TYPE "GCS7_M_FB55_Data"	// UDT 20550
VERSION : 0.0
  STRUCT
   StCode : INT ;	// State as code 32=StFault 1=StStopped 2=StStarting 3=StStartedWait 4=StStartedF
   InEnableMill1 : BOOL ;	// Enable to run mill 1
   InEnableMill2 : BOOL ;	// Enable to run mill 2
   InDischargeOkMill1 : BOOL ;	// Discharge of mill 1 is ok, starting condition
   InDischargeOkMill2 : BOOL ;	// Discharge of mill 2 is ok, starting condition
   InUsedMill1 : BOOL ;	// Mill 1 is used
   InUsedMill2 : BOOL ;	// Mill 2 is used
   InEnableFeedMill1 : BOOL ;	// Enable feeding mill 1
   InEnableFeedMill2 : BOOL ;	// Enable feeding mill 2
   CmdTick100ms : BOOL ;	// Tick 100 ms to count time (e.g. brake time)
   spare0301 : BOOL ;	//
   CmdNext : BOOL ;	// Pulse to start the next motor in automatic mode
   CmdFaultReset : BOOL ;	// Command to reset fault
   InLocal : BOOL ;	// Local mode, accept all faults
   spare0305 : BOOL ;	//
   spare0306 : BOOL ;	//
   InSeqStop : BOOL ;	// Mill will stop automatically after idling time
   OutFeedingMill1 : BOOL ;	// Mill 1 is feeding
   OutFeedingMill2 : BOOL ;	// Mill 2 is feeding
   OutLoadedMill1 : BOOL ;	// Mill 1 is loaded with product
   OutLoadedMill2 : BOOL ;	// Mill 2 is loaded with product
   OutEmptyingMill1 : BOOL ;	// Mill 1 emptying time t1 is running
   OutEmptyingMill2 : BOOL ;	// Mill 2 emptying time t2 is running
   OutEmptyingDoneMill1 : BOOL ;	// Emptying time done mill 1
   OutEmptyingDoneMill2 : BOOL ;	// Emptying time done mill 2
   StStopped : BOOL ;	// All motors are stopped
   StStarting : BOOL ;	// Not all relevant motors are started
   StStarted : BOOL ;	// All used motors are started
   StStopping : BOOL ;	// Any motor is stopping
   StFault : BOOL ;	// Any relevant element has a fault
   spare0505 : BOOL ;	//
   spare0506 : BOOL ;	//
   spare0507 : BOOL ;	//
   InBrakeMill1 : BOOL ;	// Brake mill 1
   InBrakeMill2 : BOOL ;	// Brake mill 2
   InOutRevMill : BOOL ;	// Mill motors will be started reverse
   InFastMill : BOOL ;	// Mill motors will be started fast
   spare0604 : BOOL ;	//
   spare0605 : BOOL ;	//
   spare0606 : BOOL ;	//
   spare0607 : BOOL ;	//
   InAlarmTempMill1 : BOOL ;	// Temperature alarm mill 1, changing to fault
   InAlarmTempMill2 : BOOL ;	// Temperature alarm mill 2, changing to fault
   spare0702 : BOOL ;	//
   spare0703 : BOOL ;	//
   InpS311Z2 : BOOL ;	// Digital input S311Z2: automatic mode mill 1
   InpS361Z2 : BOOL ;	// Digital input S361Z2: automatic mode mill 2
   InpS311Z2_1 : BOOL ;	// Digital input S311Z2/1: service mode mill 1
   InpS361Z2_1 : BOOL ;	// Digital input S361Z2/1: service mode mill 2
   InpS311Z3 : BOOL ;	// Digital input S311Z3: open cone mill 1
   InpS361Z3 : BOOL ;	// Digital input S361Z3: open cone mill 2
   InpS311Z4 : BOOL ;	// Digital input S311Z4: close cone mill 1
   InpS361Z4 : BOOL ;	// Digital input S361Z4: close cone mill 2
   InpS311Z5 : BOOL ;	// Digital input S311Z5: open haevy-particle gate mill 1
   InpS361Z5 : BOOL ;	// Digital input S361Z5: open haevy-particle gate mill 2
   InpS311Z6 : BOOL ;	// Digital input S311Z6: screen change acknowledge mill 1
   InpS361Z6 : BOOL ;	// Digital input S361Z6: screen change acknowledge mill 2
   OutRevMill : BOOL ;	// Mill motors are running reverse
   OutFastMill1 : BOOL ;	// Motor mill 1 is  running fast
   OutFastMill2 : BOOL ;	// Motor mill 2 is  running fast
   spare0903 : BOOL ;	//
   OutEmptyRunMill1 : BOOL ;	// Mill 1 is empty running (without product)
   OutEmptyRunMill2 : BOOL ;	// Mill 2 is empty running (without product)
   OutEmptySeqStopMill1 : BOOL ;	// Mill 1 empty running sequence stop active
   OutEmptySeqStopMill2 : BOOL ;	// Mill 2 empty running sequence stop active
   OutAlarmMill1 : BOOL ;	// Mill 1 has an alarm, any element has a fault
   OutAlarmMill2 : BOOL ;	// Mill 2 has an alarm, any element has a fault
   OutBrakeMill1 : BOOL ;	// Brake mill 1
   OutBrakeMill2 : BOOL ;	// Brake mill 2
   OutpBrakeMill1 : BOOL ;	// Digital output: brake mill 1, motor M300 has no standstill
   OutpBrakeMill2 : BOOL ;	// Digital output: brake mill 2, motor M350 has no standstill
   OutpH311Z3 : BOOL ;	// Digital output H311Z3: alarm lamp mill 1
   OutpH361Z3 : BOOL ;	// Digital output H361Z3: alarm lamp mill 2
   OutpS311Z3 : BOOL ;	// Digital output S311Z3: release for opening cone mill 1
   OutpS361Z3 : BOOL ;	// Digital output S361Z3: release for opening cone mill 2
   OutpS311Z4 : BOOL ;	// Digital output S311Z4: release for closing cone mill 1
   OutpS361Z4 : BOOL ;	// Digital output S361Z4: release for closing cone mill 2
   OutpS311Z5 : BOOL ;	// Digital output S311Z5: release for opening heavy-particle gate mill 1
   OutpS361Z5 : BOOL ;	// Digital output S361Z5: release for opening heavy-particle gate mill 2
   OutpS311Z6 : BOOL ;	// Digital output S311Z6: request for screen change mill 1
   OutpS361Z6 : BOOL ;	// Digital output S361Z6: request for screen change mill 2
   InDFCMSetpointMill1 : INT ;	// DFCM setpoint mill 1 [0.01 %]
   InDFCMSetpointMill2 : INT ;	// DFCM setpoint mill 2 [0.01 %]
   OutDFCMLoadAcMill1 : INT ;	// DFCM actual load mill 1 [0.01 %]
   OutDFCMLoadAcMill2 : INT ;	// DFCM actual load mill 2 [0.01 %]
   InScreenNoMill1 : INT ;	// Selected screen number mill 1
   InScreenNoMill2 : INT ;	// Selected screen number mill 2
   OutScreenNoAcMill1 : INT ;	// Actual screen number mill 1
   OutScreenNoAcMill2 : INT ;	// Actual screen number mill 2
   OutEmptyTimeMill1 : INT ;	// Actual time t1: emptying mill 1 [0.1 s]
   OutEmptyTimeMill2 : INT ;	// Actual time t2: emptying mill 2 [0.1 s]
   OutBrakeTimeMill1 : INT ;	// Actual time t3: braking mill 1 [0.1 s]
   OutBrakeTimeMill2 : INT ;	// Actual time t4: braking mill 2 [0.1 s]
   OutSwitchChTimeMill1 : INT ;	// Actual time t5: changing switches mill 1 [0.1 s]
   OutSwitchChTimeMill2 : INT ;	// Actual time t5: changing switches mill 2 [0.1 s]
   spare4000 : INT ;	//
   Par : STRUCT
    ParObjectNo : INT ;	// Is used for communication with PC. e.g. for message
    ParWithMill2 : BOOL ;	// With mill 2 (0= only mill 1 and its modules are used)
    ParWithFlapBox : BOOL ;	// With flap box (two-way valve)
    ParWithGateMill1 : BOOL ;	// With segment gate mill 1
    ParWithGateMill2 : BOOL ;	// With segment gate mill 2
    ParWithDFAV : BOOL ;	// With DFAV feeder / gravity separator
    ParWithDFCM : BOOL ;	// With DFCM control unit
    ParSpare0406 : BOOL ;
    ParHwDirWhileBrake : BOOL ;	// Hardware changes automatically direction while brake
    ParEmptyRunMill1 : INT ;	// Mill 1 is empty running at ? [0.01 %] load
    ParEmptyRunMill2 : INT ;	// Mill 2 is empty running at ? [0.01 %] load
    ParEmptyTimeMill1 : INT ;	// t1: Emptying time mill 1 [0.1 s]
    ParEmptyTimeMill2 : INT ;	// t2: Emptying time mill 2 [0.1 s]
    ParBrakeTimeMill1 : INT ;	// t3: Brake time mill 1 [0.1 s]
    ParBrakeTimeMill2 : INT ;	// t4: Brake time mill 2 [0.1 s]
    ParSwitchChTime : INT ;	// t5: Switch change time between slow <-> fast [0.1 s]
    spare18 : INT ;
    OutUnlockConeMill1 : BOOL ;	// Request to unlock cone mill 1
    OutUnlockConeMill2 : BOOL ;	// Request to unlock cone mill 2
    OutConeOpenedMill1 : BOOL ;	// Cone was opened for screen change mill 1
    OutConeOpenedMill2 : BOOL ;	// Cone was opened for screen change mill 2
    OutBrakeAcvMill1 : BOOL ;	// Braking is active mill 1
    OutBrakeAcvMill2 : BOOL ;	// Braking is active mill 2
    OutSwitchChMill1 : BOOL ;	// Switch changing time is active mill 1
    OutSwitchChMill2 : BOOL ;	// Switch changing time is active mill 2
    OutSwitchChDoneMill1 : BOOL ;	// Switch changing time done mill 1
    OutSwitchChDoneMill2 : BOOL ;	// Switch changing time done mill 2
    OutSpeedChMill1 : BOOL ;	// Speed changing event is active mill 1
    OutSpeedChMill2 : BOOL ;	// Speed changing event is active mill 2
    OutScreenChMill1 : BOOL ;	// Screen change is active mill 1
    OutScreenChMill2 : BOOL ;	// Screen change is active mill 2
    spare2306 : BOOL ;
    OutInPosFlapBox : BOOL ;	// Flap box is in correct position
   END_STRUCT ;
  END_STRUCT ;	
END_TYPE

TYPE "GCS7_M_FB56_Data"	// UDT 20560
VERSION : 0.0
  STRUCT 	// Interface to maschine FB50
   StCode : INT ;	//State as code
   InEnable : BOOL ;	//Enable to run the motor reverse
   InRestDischarge : BOOL ;	//Rest discharge of the bin
   InDisableVibro : BOOL ;	//Disable Vibro
   InUncovered : BOOL ;	//Low Level Bin is uncovered : Condition for OutUncovered
   InCovered : BOOL ;	//Low Level Bin is covered   : Condition for Vibro
   spare0205 : BOOL ;
   spare0206 : BOOL ;
   spare0207 : BOOL ;
   CmdOff : BOOL ;	//Pulse to start the element immediately (manual mode)
   CmdOn : BOOL ;	//Pulse to stop  the element immediately (manual mode)
   CmdNext : BOOL ;	//Pulse to start the element in automatic mode
   CmdFaultReset : BOOL ;	//Command to reset fault
   InLocal : BOOL ;	//1= Local mode (no fault by start with service switch)
   InManual : BOOL ;	//1= Manual/ 0=Automatic
   spare0306 : BOOL ;
   spare0307 : BOOL ;
   OutUncovered : BOOL ;	//Low level is unvovered
   OutRestDischarged : BOOL ;	//Bin is rest discharged
   OutEmpty : BOOL ;	//Relevant level: uncovered or rest discharged
   OutPulseVibroOn : BOOL ;	//Command to start vibro
   OutEdgeFlowCovered : BOOL ;
   spare0405 : BOOL ;
   spare0406 : BOOL ;
   spare0407 : BOOL ;
   StStopped : BOOL ;	//Motor is stopped
   StStarting : BOOL ;	//Motor is starting
   StStarted : BOOL ;	//Motor is started
   StStopping : BOOL ;	//Motor is stopping
   StFault : BOOL ;	//Machine has a fault
   Par : STRUCT
    ParObjectNo : INT ;	//Is used for communication with PC
    ParWithVibro : BOOL ;	//With element
    ParWithLL : BOOL  := TRUE;	//With element
    ParWithFlow : BOOL  := TRUE;	//With element flow detector
    ParDischargerIsMotor : BOOL ;	//Discharger is Motor
    ParContinuous : BOOL ;	//Vibro is running continuous if discharger is started
    ParVibroOnTime : INT ;	//Length pulse on (t1)
    ParVibroOffTime : INT ;	//Length pulse off (t2)
    ParRestDischargeTime : INT ;	//Time until bin is completly discharged
    OutDelayTime : INT ;	//Actual time t1 or t2
    OutRestDischargeTime : INT ;
    spare16 : INT ;
   END_STRUCT ;
  END_STRUCT ;	
END_TYPE

TYPE "GCS7_M_FB58_Data"	// UDT 20580
VERSION : 0.1
  STRUCT
   StCode : INT ;	//Element state code
   InEnable : BOOL ;	//Enable to run the element reverse
   InEngage : BOOL ;	//Enable to run engage
   InNewJobWait : BOOL ;	//Signal to wait for Start Job Change from the Operator
   InFeedRoll : BOOL ;
   spare24 : BOOL ;
   CmdNewJob : BOOL ;	//Pulse to start the element in automatic mode (see global flags)
   spare26 : BOOL ;
   spare27 : BOOL ;
   CmdOff : BOOL ;	//Pulse to stop the element immediately (manual mode)
   CmdOn : BOOL ;	//Pulse to start the element immediately (manual mode)
   CmdNext : BOOL ;	//Pulse to start the element in automatic mode (see global flags)
   CmdFaultReset : BOOL ;	//Command to reset fault
   InLocal : BOOL ;	//1= Local mode (no fault by start with service switch)
   InManual : BOOL ;	//1= Manual/ 0=Automatic
   InReport : BOOL ;	//Report of all state transitions
   InSeqStop : BOOL ;	//Stop automatically after idling time
   spare40 : BOOL ;
   spare41 : BOOL ;
   InSimulation : BOOL ;	//DP:
   OutComFault : BOOL ;	//Communication fault
   spare44 : BOOL ;
   spare45 : BOOL ;
   spare46 : BOOL ;
   OutWarning : BOOL ;	//Warning
   StStopped : BOOL ;	//BCFA in state Automatic.Stopped
   StStarting : BOOL ;	//BCFA in state Automatic.Starting
   StProduction : BOOL ;	//BCFA in state Automatic.Production
   StStopping : BOOL ;	//BCFA in state Automatic.Stopping
   StFaultCom : BOOL ;
   StStandby : BOOL ;	//BCFA in state Automatic.Standby
   StService : BOOL ;	//BCFA is in mode Servive or Neutral
   OutFaulted : BOOL ;	//Fault
   ToBCFA : STRUCT
    SP_GapLeft : INT ;	//Setpoint gap left
    SP_GapRight : INT ;	//Setpoint gap right
    SP_TempRoll : INT ;	//Setpoint water temperture
    SP_FE_RollSpeed : INT ;	//Setpoint speed roll feeder
    SP_FE_VibroSpeed : INT ;	//Setpoint speed vibro feeder
    SP_RC_Option : INT ;	//Setpoint roll cooling option (1 = with, 2 = without)
    res120 : INT ;
    res140 : INT ;
    res160 : INT ;
    res180 : INT ;
    CmdSequenceStart : BOOL ;	//Start flaker
    CmdSequenceStop : BOOL ;	//Sequence stop flaker
    CmdReleaseEngage : BOOL ;	//Plant release signal (=> E0.0) (e.q. release roll engage on site)
    CmdDoneJobchange : BOOL ;	//Job change executed
    CmdReleaseFeed : BOOL ;
    res205 : BOOL ;
    res206 : BOOL ;
    res207 : BOOL ;
    res210 : BOOL ;
    res211 : BOOL ;
    res212 : BOOL ;
    res213 : BOOL ;
    res214 : BOOL ;
    res215 : BOOL ;
    res216 : BOOL ;
    res217 : BOOL ;
    res220 : WORD ;
    res240 : WORD ;
    res260 : WORD ;
    res280 : WORD ;
    LineCheck : WORD ;	//Line check value from remote
   END_STRUCT ;
   FromBCFA1 : STRUCT
    RV_GapLeft : INT ;	//Actual gap value left
    RV_GapRight : INT ;	//Actual gap value right
    RV_TempRoll : INT ;	//Actual water temperature
    RV_MM_1_Current : INT ;	//Actual current mainmotor 1
    RV_MM_2_Current : INT ;	//Actual current mainmotor 2
    RV_ForceLeft : INT ;	//Actual roll force left
    RV_ForceRight : INT ;	//Actual roll force right
    RV_FE_DSDC_Temp : INT ;	//Actual conditioner temperature
    res480 : INT ;
    RV_SP_GapLeft : INT ;	//Actual setpoint gap left
    RV_SP_GapRight : INT ;	//Actual setpoint gap right
    RV_SP_TempRoll : INT ;	//Actual setpoint water temperture
    RV_SP_FE_RollSpeed : INT ;	//Actual setpoint speed roll feeder
    RV_SP_FE_VibroSpeed : INT ;	//Actual setpoint speed vibro feeder
    RV_SP_RC_Option : INT ;	//Actual setpoint roll cooling option (1 = with, 2 = without)
    res620 : INT ;
   END_STRUCT ;
   FromBCFA2 : STRUCT
    Sta_Automatic : BYTE ;	//Status automatic mode
    Sta_Calibration : BYTE ;	//Status calibration mode
    Sta_OperationMode : BYTE ;	//Status operation mode
    Sta_MM_1_On : BOOL ;	//Mainmotor 1 running
    Sta_MM_1_Fault : BOOL ;	//Mainmotor 1 fault
    Sta_MM_2_On : BOOL ;	//Mainmotor 2 running
    Sta_MM_2_Fault : BOOL ;	//Mainmotor 2 fault
    Sta_ROLL_On : BOOL ;	//Roll feeder running
    Sta_ROLL_Fault : BOOL ;	//Roll feeder fault
    Sta_Vibro_On : BOOL ;	//Vibro channel running
    Sta_Vibro_Fault : BOOL ;	//Vibro cahnnel fault
    Sta_RC_On : BOOL ;	//Roll cooling on
    Sta_RC_Fault : BOOL ;	//Roll cooling fault
    Sta_HD_On : BOOL ;	//Hydraulic running
    Sta_HD_Fault : BOOL ;	//Hydraulic fault
    Sta_Engaged_On : BOOL ;	//Roll position engaged
    Sta_Engaged_Fault : BOOL ;	//Roll position fault
    Sta_Flap_Production : BOOL ;	//Outlet flap production (DSDC option)
    Sta_Flap_Fault : BOOL ;	//Outlet flap fault (DSDC option)
    res690 : BYTE ;
    res700 : WORD ;
    res702 : WORD ;
    CmdStartJobchange : BOOL ;	//Start job change
    res741 : BOOL ;
    res742 : BOOL ;
    res743 : BOOL ;
    res744 : BOOL ;
    res745 : BOOL ;
    res746 : BOOL ;
    res747 : BOOL ;
    res750 : BYTE ;
    Alarm : STRUCT 	//Aux. signal to retry fault message
     A01System : BOOL ;
     A02Memory : BOOL ;
     A03SerialCom : BOOL ;
     A04MainMotor : BOOL ;
     A05MMotor1Range : BOOL ;
     A06MMotor2Range : BOOL ;
     A07Hydraulic : BOOL ;
     A08HydrPressTOut : BOOL ;
     A09 : BOOL ;
     A10GapAdjMotor : BOOL ;
     A11GapLeftEdpos : BOOL ;
     A12GapLeftRange : BOOL ;
     A13GapRightEndpos : BOOL ;
     A14GapRightRange : BOOL ;
     A15 : BOOL ;
     A16DryRunning : BOOL ;
     A17ProductNokWA : BOOL ;
     A18ProductNokAL : BOOL ;
     A19FeederMotor : BOOL ;
     A20WaterFlow : BOOL ;
     A21RollTpWA : BOOL ;
     A22RollTpMax : BOOL ;
     A23WaterTpRange : BOOL ;
     A24CondTpMinWA : BOOL ;
     A25CondTpMinAL : BOOL ;
     A26AirPressure : BOOL ;
     A27CondTpRange : BOOL ;
     A28ForceLeftRange : BOOL ;
     A29ForceRightRange : BOOL ;
     A30 : BOOL ;
     A31ProtectionKnife : BOOL ;
     A32ProtectionCover : BOOL ;
    END_STRUCT ;
    Message : DWORD ;
    res840 : WORD ;
    res860 : WORD ;
    res880 : WORD ;
    res900 : WORD ;
    res920 : WORD ;
    LineCheck : WORD ;	//Line check value to remote
   END_STRUCT ;
   OutAlarmNr : INT ;	//Is read from MEAF ; Is transformed for MWEB like MEAF
   OutAlarmNrLog : INT ;	//Last textnumber send to log
   Par : STRUCT
    ParObjectNo : INT ;	//Is used for communication with PC, e.g. for message
    ParMsgType : INT ;	//Is used for message (translation of state)
    ParHornCode : INT ;	//Is used by horn module
    ParLogOff : BOOL ;	//Report is off
    ParManual : BOOL ;	//Manual mode without interlocking
    ParIOByteNr : INT ;	//Address of first input and output byte
    ParSpare : INT ;
    CopyData : STRUCT
     Alarm : DWORD ;
     SP_GapLeft : INT ;	//Setpoint gap left
     SP_GapRight : INT ;	//Setpoint gap right
     SP_TempRoll : INT ;	//Setpoint water temperture
     SP_FE_RollSpeed : INT ;	//Setpoint speed roll feeder
     SP_FE_VibroSpeed : INT ;	//Setpoint speed vibro feeder
     SP_RC_Option : INT ;	//Setpoint roll cooling option (1 = with, 2 = without)
     res120 : INT ;
     res140 : INT ;
    END_STRUCT ;
    OutHelpFlags : STRUCT 	//Aux. signal to retry fault message
     OutComFaultRead : BOOL ;
     OutComFaultSend : BOOL ;
     OutFaultedMsg : BOOL ;
     OutComFaultMsg : BOOL ;
    END_STRUCT ;
   END_STRUCT ;
  END_STRUCT ;	
END_TYPE

TYPE "GCS7_M_FB59_Data"	// UDT 20590
VERSION : 0.0
  STRUCT 	// Interface to maschine FB50
   StCode : INT ;	//State as code
   InEnable : BOOL ;	//Enable to run the motor reverse
   InRestDischarge : BOOL ;	//Rest discharge of the bin
   InMonLSFault : BOOL ;	//Fault if flap maximum open (indempendend of state of LL)
   InUncovered : BOOL ;	//LL is uncovered
   InCovered : BOOL ;	//LL is covered
   CmdNewJob : BOOL ;	//Command new job
   spare0206 : BOOL ;
   spare0207 : BOOL ;
   CmdOff : BOOL ;	//Pulse to start the element immediately (manual mode)
   CmdOn : BOOL ;	//Pulse to stop  the element immediately (manual mode)
   CmdNext : BOOL ;	//Pulse to start the element in automatic mode
   CmdFaultReset : BOOL ;	//Command to reset fault
   InLocal : BOOL ;	//1= Local mode (no fault by start with service switch)
   InManual : BOOL ;	//1= Manual/ 0=Automatic
   spare0306 : BOOL ;
   spare0307 : BOOL ;
   spare0400 : BOOL ;
   spare0401 : BOOL ;
   OutEmpty : BOOL ;	//Bin is rest discharged
   spare0403 : BOOL ;
   spare0404 : BOOL ;
   spare0405 : BOOL ;
   spare0406 : BOOL ;
   spare0407 : BOOL ;
   StStopped : BOOL ;
   StStarting : BOOL ;
   StStarted : BOOL ;
   StStopping : BOOL ;
   StFault : BOOL ;
   StWaiting : BOOL ;	//Waiting for product flow
   Par : STRUCT
    ParObjectNo : INT ;	//Is used for communication with PC
    ParWithLL : BOOL  := TRUE;	//With element
    spare6 : INT ;
    spare8 : INT ;
    spare10 : INT ;
   END_STRUCT ;
  END_STRUCT ;	
END_TYPE

TYPE "GCS7_M_FB60_Data"	// UDT 20600
VERSION : 0.0
  STRUCT 	// Interface to maschine FB50
   StCode : INT ;	//State as code
   InEnable : BOOL ;	//Enable to run aspiration (0=Airlock stops after idling time)
   InDisableAirlock : BOOL ;	//Immediately stop of Airlock
   InDisableFilter : BOOL ;	//Immediately stop Filter controller
   InDisableDischarger : BOOL ;	//Immediately stop Discharger
   spare04 : BOOL ;
   spare05 : BOOL ;
   spare06 : BOOL ;
   spare07 : BOOL ;
   CmdOffMan : BOOL ;	//Pulse to stop all elements immediately (manual mode)
   CmdOnMan : BOOL ;	//Pulse to start  the next element (manual mode)
   CmdNext : BOOL ;	//Pulse to start the element in automatic mode (see global flags)
   CmdFaultReset : BOOL ;	//Command to reset fault
   InLocal : BOOL ;	//1= Local mode (no fault by start with service switch)
   InManual : BOOL ;	//1= Manual/ 0=Automatic
   CmdFanOffMan : BOOL ;	//Pulse to stop the Fan in manual mode
   InSeqStop : BOOL ;	//Stop automatically after idling time
   OutWarning : BOOL ;	//Pressure to high
   spare0201 : BOOL ;
   spare0202 : BOOL ;
   OutPulseVibroOn : BOOL ;	//Internal used for pulsing
   spare0204 : BOOL ;
   spare0205 : BOOL ;
   spare0206 : BOOL ;
   spare0207 : BOOL ;
   StStopped : BOOL ;	//Aspiration is stopped
   StStarting : BOOL ;	//Fan or Airlock is starting
   StStarted : BOOL ;	//Fan and Airlock are started
   StStopping : BOOL ;	//Fan is stopping
   StFault : BOOL ;	//Any element is in state StFault
   StIdling : BOOL ;	//Idling time of Airlock is running
   Par : STRUCT
    ParObjectNo : INT ;	//Is used for communication with PC
    ParWithAirlock : BOOL ;	//Machine uses this element
    ParWithFan : BOOL ;	//Machine uses this element
    ParWithFilter : BOOL ;	//Machine uses this element
    ParWithARF : BOOL ;	//Machine uses this element
    ParWithLSDoor : BOOL ;	//Machine uses this element
    ParWithPressure : BOOL ;	//Machine uses this element
    ParWithHLAirlock : BOOL ;	//Machine uses this element
    ParWithDischarger : BOOL ;	//Machine uses this element
    ParVibroOnTime : INT ;	//Length pulse on (t1)
    ParVibroOffTime : INT ;	//Length pulse off (t2)
    OutDelayTime : INT ;	//Actual time t1 or t2
    spare1 : INT ;
    spare2 : INT ;
   END_STRUCT ;
  END_STRUCT ;	
END_TYPE

TYPE "GCS7_M_FB61_Data"	// UDT 20610
VERSION : 0.0
  STRUCT 	// Interface to maschine FB50
   StCode : INT ;	//State as code
   InEnable : BOOL ;	//Enable to run the machine
   spare0201 : BOOL ;
   InDisableAirlock : BOOL ;	//Stop airlock
   spare0203 : BOOL ;
   CmdNewValue : BOOL ;	//Command send new value to scale
   CmdNewJob : BOOL ;	//Command new job
   spare0206 : BOOL ;
   InOutEmptyingHopperScale : BOOL ;	//Emptying scale and hopper above scale
   CmdOff : BOOL ;	//Pulse to start the element immediately (manual mode)
   CmdOn : BOOL ;	//Pulse to stop  the element immediately (manual mode)
   CmdNext : BOOL ;	//Pulse to start the element in automatic mode
   CmdFaultReset : BOOL ;	//Command to reset fault
   InLocal : BOOL ;	//1= Local mode (no fault by start with service switch)
   InManual : BOOL ;	//1= Manual/ 0=Automatic
   spare0306 : BOOL ;
   InSeqStop : BOOL ;	//Stop automatically after idling time
   OutStopPoint : BOOL ;	//Target weight reached
   OutEmptyOutlet : BOOL ;	//HL Outlet uncovered
   OutEmptyInlet : BOOL ;	//LL Inlet uncovered
   spare0403 : BOOL ;
   spare0404 : BOOL ;
   spare0405 : BOOL ;
   spare0406 : BOOL ;
   spare0407 : BOOL ;
   StStopped : BOOL ;
   StStarting : BOOL ;
   StStarted : BOOL ;
   StStopping : BOOL ;
   StFault : BOOL ;
   StWaiting : BOOL ;
   StEmptying : BOOL ;
   StEmptied : BOOL ;
   Par : STRUCT
    ParObjectNo : INT ;	//Is used for communication with PC
    ParWithAirlock : BOOL ;	//With element Airlock
    ParWithLLOutlet : BOOL ;	//With element LLOutlet
    ParWithHLInlet : BOOL ;	//With element HLInlet
    ParStopAirlockByLL : BOOL ;	//Stop airlock if LLOutlet is uncovered
    ParHLOutletLocal : BOOL ;	//No HLOutlet fault, element is in local mode
   END_STRUCT ;
  END_STRUCT ;	
END_TYPE

TYPE "GCS7_M_FB62_Data"	// UDT 20620
VERSION : 0.0
  STRUCT 	// Interface to maschine FB50
   StCode : INT ;	//State as code
   InEnable : BOOL ;	//Enable to run the motor
   InReleaseOutput : BOOL ;	//Enable to release Output
   InFeeding : BOOL ;	//Feed is started
   InMonFault : BOOL ;	//1=Fault, 0=Warning
   InClearing : BOOL ;	//Stop motor after Clearing time
   spare0205 : BOOL ;
   spare0206 : BOOL ;
   spare0207 : BOOL ;
   CmdOff : BOOL ;	//Pulse to stop the machine in manual mode
   CmdOn : BOOL ;	//Pulse to start machine in manual mode
   CmdNext : BOOL ;	//Pulse to start the element in automatic mode
   CmdFaultReset : BOOL ;	//Command to reset fault
   InLocal : BOOL ;	//1= Local mode (no fault by start with service switch)
   InManual : BOOL ;	//1= Manual/ 0=Automatic
   spare16 : BOOL ;
   InSeqStop : BOOL ;	//Stop automatically after idling time
   spare0400 : BOOL ;
   OutLoaded : BOOL ;
   OutMonitoring : BOOL ;	//Monitoring is active
   OutWarning : BOOL ;	//Warning mode of Analog Signal
   spare0404 : BOOL ;
   spare0405 : BOOL ;
   spare0406 : BOOL ;
   spare0407 : BOOL ;
   StStopped : BOOL ;	//Motor is stopped
   StStarting : BOOL ;	//Motor is starting
   StStarted : BOOL ;	//Motor is started
   StStopping : BOOL ;	//Motor is stopping
   StFault : BOOL ;	//Machine has a fault
   StClearing : BOOL ;	//Clearing time is running
   StDosing : BOOL ;	//Motor ist started and Output is released
   Par : STRUCT
    ParObjectNo : INT ;	//Is used for communication with PC
    ParWithMon1 : BOOL  := TRUE;	//With element Mon1
    ParWithRelease : BOOL  := TRUE;	//With element Release
    ParClearingTime : INT ;	//Clearing time by deselect motor befor stop
    ParDelayRelease : INT ;	//Starting Delay RelaseOutput
    ParCurrentNom : INT ;	//Nominal Current of Drive [A]
    ParLimitMin : INT ;	//Minimum Limit of current of drive [%]
    ParLimitMax : INT ;	//Maximum limit of current of drive [%]
    spare14 : INT ;
    OutClearingTime : INT ;	//Actual clearing time
    OutDelayDosing : INT ;	//Actual starting delay time
    spare20 : INT ;
   END_STRUCT ;
  END_STRUCT ;	
END_TYPE

TYPE "GCS7_M_FB63_Data"	// UDT 20630
VERSION : 0.0
  STRUCT 	// Parameter for maschine FB50
   StCode : INT ;	//machine state code
   InEnable : BOOL ;	//-->de:"Start Presse"
   InDischargerRunning : BOOL ;	//-->de:"Abtransport läuft"
   InSuspend : BOOL ;	//-->de:"Dosierunterbruch"
   InOutCoolerOnMan : BOOL ;	//-->de:"Austrag Gegenstromkühler manuell ein"
   InOutHeaterOnMan : BOOL ;	//-->de:"Pressenheizung manuell ein"
   CmdNewJob : BOOL ;	//-->de:"Reset Mehlmenge"
   InOverrideLLHopper : BOOL ;	//-->de:"Ueberbrueckung Vordepot Leerstand"
   spare0207 : BOOL ;
   CmdOff : BOOL ;	//Pulse to stop the machine immediately (manual mode)
   CmdOn : BOOL ;	//Pulse to start the machine (manual mode)
   CmdNext : BOOL ;	//Pulse to start the machine in automatic mode (see global flags)
   CmdFaultReset : BOOL ;	//-->de:"Reset alle Alarme"
   InLocal : BOOL ;	//1= Local mode (no fault by start with service switch)
   InManual : BOOL ;	//1= Manual / 0= Automatic: Set and reset by PC
   CmdResetHorn : BOOL ;	//--> de:"Reset Horn"
   InRemoteMode : BOOL ;	//Remote Mode selected by Host
   CmdSendB101 : BOOL ;	//--> Send telegramm B101 to DFCA: Set values
   CmdSendB102 : BOOL ;	//--> Send telegramm B102 to DFCA: Form name recipe ident
   CmdSendB103 : BOOL ;	//--> Send telegramm B103 to DFCA: Recipe name
   InpLL : BOOL ;	//DI (all types): Low Level Brain Bin    -->OutpLL  (1=Covered)
   InpLevelMiddle : BOOL ;	//DI (all types): Middle Level Brain Bin -->OutpLevelMiddle (1=Covered)
   CmdSendB104 : BOOL ;	//--> Send telegramm B104 to DFCB, DFBB: RecipeGroup
   InOutFanOnMan : BOOL ;	//-->de:"Vetilator Heisluft manuell ein"
   spare0407 : BOOL ;
   StIdle : BOOL ;	//DFCA: Mode en: Idle position / pre-start        de: Ruhestellung/Vorstart
   StStartup : BOOL ;	//DFCA: Mode en: Start-Up                         de: Anfahren
   StReady : BOOL ;	//DFCA: Mode en: Feed readiness /Feed interrupted de: Dosierbereitschaft
   StFeedStartup : BOOL ;	//DFCA: Mode en: Feed start-up                    de: Dosierstart
   StFault : BOOL ;	//DFCA: InpSumFault is on
   StOperation : BOOL ;	//DFCA: Mode en: Operation                        de: Betrieb
   StShutdown : BOOL ;	//DFCA: Mode en: Shutdown                         de: Stoppen
   spare57 : BOOL ;
   OutpLL : BOOL ;	//<--Dig. Output to DFCA  (all types): de:Leerstand Kleiesilo (1=Covered)
   OutpLevelMiddle : BOOL ;	//<--Dig. Output to DFCA  (all types): de:Mittelstand Kleiesilo (1=Covered)
   OutpLampRunning : BOOL ;	//<--Dig. Output to Relay control: Signallampe Betrieb
   OutpLampFault : BOOL ;	//<--Dig. Output to Relay control: Signallampe Störung
   OutpLampFireAlarm : BOOL ;	//<--Dig. Output to Relay control: Signallampe Brandschutzalarm
   Par : STRUCT
    ParObjectNo : INT ;	//Is used for communication with PC
    ParDP : BOOL  := TRUE;	//With DP connection
    ParManual : BOOL  := TRUE;	//Manual mode without interlocking
    ParSpare1 : BOOL ;
    ParSpare04 : BOOL ;
    ParIOByteNr : INT ;	//Byte Address DP
    ParFaultResetTime : INT  := 20;	//[0.1s]
    OutFaultResetTime : INT ;	//[0.1s]
    Spare12 : INT ;
   END_STRUCT ;
  END_STRUCT ;	
END_TYPE

TYPE "GCS7_M_FB64_Data"	// UDT 20640
VERSION : 0.0
  STRUCT 	// Interface to maschine FB50
   StCode : INT ;	//State as code
   InEnable : BOOL ;	//Enable to run the machine, discharge ok
   InProductFeed : BOOL ;	//Signal product feed
   InDisableWaterDosing : BOOL ;	//Immediate stop water dosing
   InDisableConveyor : BOOL ;	//Interlocking with HL
   CmdNewValue : BOOL ;	//Send new target value to MYEB
   CmdNewJob : BOOL ;	//Clear actual values of MYEB
   spare0206 : BOOL ;
   spare0207 : BOOL ;
   CmdOff : BOOL ;	//Pulse to stopp the element immediately (manual mode)
   CmdOn : BOOL ;	//Pulse to start  the element immediately (manual mode)
   CmdNext : BOOL ;	//Pulse to start the element in automatic mode (see global flags)
   CmdFaultReset : BOOL ;	//Command to reset fault
   InLocal : BOOL ;	//1=Local mode (no fault by start with service switch)
   InManual : BOOL ;	//1=Manual/ 0=Automatic
   InLocalWaterControl : BOOL ;	//1=Local Water Control
   InManualWaterControl : BOOL ;	//1=Manual controled water / 0=Automatic
   OutOffDelayFeedRun : BOOL ;	//Aux. signal switch off delay feed is running
   OutOffDelayFeedDone : BOOL ;	//Aux. signal switch off delay feed done
   OutOnDelayWaterRun : BOOL ;	//Aux. signal switch on delay water is running
   OutOnDelayWaterDone : BOOL ;	//Aux. signal switch on delay water done
   OutMoistureStartPc : BOOL ;	//Aux. signal moisture start with [%] factor
   OutMoistureStart : BOOL ;	//Aux. signal moisture start
   spare0406 : BOOL ;
   OutFeedReady : BOOL ;	//Aux. signal machine ready for feeding
   StStopped : BOOL ;	//Machine is stopped
   StStarting : BOOL ;	//Machine is starting
   StStarted : BOOL ;	//Machine is started
   StStopping : BOOL ;	//Machine is stopping
   StFault : BOOL ;	//Machine has a fault
   Par : STRUCT
    ParObjectNo : INT ;	//Is used for communication with PC
    ParWithMYEB_LC : BOOL  := TRUE;	//With MYEB control unit MYEB_LC
    ParWithMYEB_GroupAlarm : BOOL ;	//With digital input MYEB_GroupAlarm
    ParWithMYF_Conveyor : BOOL  := TRUE;	//With digital output MYF_ConveyorEnable
    ParStartValuePc : INT ;	//Start value factor for moisture start [%]
    ParStartValue : DINT ;	//Start value for moisture start  [0.1 l/h]
    ParOffDelayFeed : INT ;	//Switch off delay after feed [0.1 s]
    ParOnDelayWater : INT ;	//Switch on delay for water   [0.1 s]
    OutOffDelayFeed : INT ;	//Actual time: off delay feed timer
    OutOnDelayWater : INT ;	//Actual time: on delay water timer
    spare18 : INT ;
    spare20 : INT ;
    spare22 : INT ;
   END_STRUCT ;
  END_STRUCT ;	
END_TYPE

TYPE "GCS7_M_FB65_Data"	// UDT 20650
VERSION : 0.0
  STRUCT 	// Interface to maschine FB50
   StCode : INT ;	//State as code
   InEnable : BOOL ;	//Enable to run machine, 0=Immediate stop
   InAirOk : BOOL ;
   spare0202 : BOOL ;
   CmdAirlockOnOff : BOOL ;	//Manual mode: Toggle
   CmdOpenAll : BOOL ;	//Manual mode:
   CmdPulsingOnOff : BOOL ;	//Manual mode: Toggle
   InClearing : BOOL ;
   InDisableAirlock : BOOL ;	//Stop airlock automatic mode
   CmdOff : BOOL ;	//Pulse to stop all elements immediately (manual mode)
   CmdMainOnOff : BOOL ;	//Manual mode: Toggle main valve
   CmdNext : BOOL ;	//Pulse to start the element in automatic mode (see global flags)
   CmdFaultReset : BOOL ;	//Command to reset fault
   InLocal : BOOL ;	//1= Local mode (no fault by start with service switch)
   InManual : BOOL ;	//1= Manual/ 0=Automatic
   InNotClearingBypass : BOOL ;	//Stopping without opening bypass valve
   spare0307 : BOOL ;	//Stop automatically after idling time
   OutManOpenAll : BOOL ;	//Manual mode: Function all flap open is selected
   OutManPulsing : BOOL ;	//Manual mode: Function pulsing is selected
   spare0402 : BOOL ;	//Any element has a fault
   spare0403 : BOOL ;
   OutFault : BOOL ;	//Summary fault
   OutLoaded : BOOL ;	//Loaded with product
   spare0406 : BOOL ;
   spare0407 : BOOL ;
   StStopped : BOOL ;
   StStarting : BOOL ;
   StStarted : BOOL ;
   StStopping : BOOL ;
   spare0504 : BOOL ;
   StClearing : BOOL ;
   StFeeding : BOOL ;
   InClearingCycles : INT ;	//(*1) Total number of requested clearings cycles
   InClearingPulses : INT ;	//(*1) Total number of requested pluses or ClearingValve per clearing cycle
   OutCntClearingCycles : INT ;	//(*1) Actual counter clearing cycles
   OutCntClearingPulse : INT ;	//(*1) Actual counter clearing pulses
   spare14 : INT ;
   spare16 : INT ;
   OutSubState : INT ;	//Substate Internal used
   Par : STRUCT
    ParObjectNo : INT ;	//Is used for communication with PC
    ParWithMainValve : BOOL ;	//With element
    ParWithMatValve : BOOL ;	//With element
    ParWithAirValve : BOOL ;	//With element
    ParWithBypassValve : BOOL ;	//With element
    ParWithSpeedMon : BOOL ;	//With element
    ParWithHL : BOOL ;	//With element
    ParWithClearingValve : BOOL ;	//With element
    ParDelayMain : INT  := 100;
    ParDelayAirlock : INT  := 100;
    ParPulseMatTime : INT  := 100;
    ParPulseAirTime : INT  := 100;	//
    ParClearingPulsing : INT  := 100;	//Clearing time : MatValve and AirValve are pulsing
    ParClearingBoth : INT  := 100;	//Cearing time  : MatValve and AirValve are open
    ParClearingBypass : INT  := 100;	//Cearing time  : BypassValve (MainValve) is open
    ParDelayClosing : INT  := 100;	//Closing delay MatValve after closing MainValev
    ParClearingValvePulseOn : INT ;	//(*1) Clearing Time : Clearing Valve pusling: Pulse Time On
    ParClearingValvePulseOff : INT ;	//(*1) Clearing Time : Clearing Valve pusling: Pulse Time Off
    ParClearing1stCycle : INT ;	//(*1) Clearing Time 1st Cycle: (ClearingValve and MatValve open)
    ParClearing2ndCycle : INT ;	//(*1) Clearing Time 2nd Cycle: (ClearingValve and MatValve open)
    ParClearingBypassAirlock : INT ;	//(*1) Clearing Time: ClearingValve=open , MatValve=closed , AirValve=open
    OutDelayTime : INT ;
    OutPulseTime : INT ;
    OutClearingTime : INT ;	//Actual total cleaing time
    OutPulseMat : BOOL ;	//Timer ParPulseMat is on
    OutDelayMainValveEnd : BOOL ;
    OutDelayAirlockEnd : BOOL ;
    OutEnableMan : BOOL ;
    OutEnableClearingValve : BOOL ;	//Internal used
    OutEnableMatValve : BOOL ;	//Internal used
    OutEnableAirValve : BOOL ;	//Internal used
    OutEnableBypassValve : BOOL ;	//Internal used
    OutClearingTimeSubstate : INT ;	//Actual clering time substate
    spare40 : INT ;
    spare42 : INT ;
    spare44 : INT ;
    spare46 : INT ;
    spare48 : INT ;
   END_STRUCT ;
  END_STRUCT ;	
END_TYPE

TYPE "GCS7_M_FB66_Data"	// UDT 20660
VERSION : 0.0
  STRUCT 	// Interface to maschine FB50
   StCode : INT ;	//State as code
   InEnable : BOOL ;	//Enable to run
   spare0201 : BOOL ;
   InBlowerStarted : BOOL ;	//External blower started
   spare0203 : BOOL ;
   spare0204 : BOOL ;
   spare0205 : BOOL ;
   InClearing : BOOL ;	//Stop Airlock
   InBlowOff : BOOL ;	//Open blow off valve (way not ok)
   CmdOff : BOOL ;	//Pulse to stop all elements immediately (manual mode)
   CmdOn : BOOL ;	//Pulse to start  the next element (manual mode)
   CmdNext : BOOL ;	//Pulse to start the element in automatic mode (see global flags)
   CmdFaultReset : BOOL ;	//Command to reset fault
   InLocal : BOOL ;	//1= Local mode (no fault by start with service switch)
   InManual : BOOL ;	//1= Manual/ 0=Automatic
   CmdAirlockOff : BOOL ;	//Pulse to stop teh Airlock (manual mode)
   InSeqStop : BOOL ;	//Stop automatically after idling time
   OutWarning : BOOL ;	//Maximum clearing time reached
   OutEnableBlower : BOOL ;	//Interlocking for external blower
   InNoWaitMinP : BOOL ;	//Not waiting for minimum pressure during clearing
   spare0403 : BOOL ;
   spare0404 : BOOL ;
   spare0405 : BOOL ;
   spare0406 : BOOL ;
   spare0407 : BOOL ;
   StStopped : BOOL ;	//Motor is stopped
   StStarting : BOOL ;	//Motor is starting
   StStarted : BOOL ;	//Motor is started forward: Next Element can start
   StStopping : BOOL ;	//Motor is stopping
   StFault : BOOL ;	//Machine has a fault
   StClearing : BOOL ;	//Clearing time running, Blower started
   StCleared : BOOL ;	//Clearing time end, Blower is started
   Par : STRUCT
    ParObjectNo : INT ;	//Is used for communication with PC
    ParWithBlowOff : BOOL ;	//With blow off valve
    ParWithHLInlet : BOOL ;	//With HL inlet
    ParBlowerExternal : BOOL ;	//Blower is erternal
    ParClearingTime : INT ;	//Clearing time target [0.1s]
    OutClearingTime : INT ;	//Actual clearing time [0.1s]
    spare : DINT ;	//
   END_STRUCT ;
  END_STRUCT ;	
END_TYPE

TYPE "GCS7_M_FB67_Data"	// UDT 20670
VERSION : 0.0
  STRUCT 	// Interface to maschine FB50
   StCode : INT ;	//State as code
   InEnable : BOOL ;	//Enable to run
   InWayB : BOOL ;
   InBlowerStarted : BOOL ;	//External blower started
   InWayAB : BOOL ;	//Open both way (only 2 lines)
   InDisableAirlockA : BOOL ;	//Stop Airlock A
   InDisableAirlockB : BOOL ;	//Stop Airlock B
   InClearing : BOOL ;	//Stop Airlock A and B, Change to clearing
   InBlowOff : BOOL ;	//Open blow off valve (way not ok)
   CmdOff : BOOL ;	//Pulse to stop all elements immediately (manual mode)
   CmdOn : BOOL ;	//Pulse to start  the next element (manual mode)
   CmdNext : BOOL ;	//Pulse to start the element in automatic mode (see global flags)
   CmdFaultReset : BOOL ;	//Command to reset fault
   InLocal : BOOL ;	//1= Local mode (no fault by start with service switch)
   InManual : BOOL ;	//1= Manual/ 0=Automatic
   CmdAirlockOff : BOOL ;	//Pulse to stop the Airlocks (manual mode)
   InSeqStop : BOOL ;	//Stop automatically after idling time
   OutWarning : BOOL ;	//Maximum clearing time reached
   OutEnableBlower : BOOL ;	//Interlocking for external blower
   InNoWaitMinP : BOOL ;	//Not waiting for minimum pressure during clearing
   spare0403 : BOOL ;
   spare0404 : BOOL ;
   spare0405 : BOOL ;
   spare0406 : BOOL ;
   spare0407 : BOOL ;
   StStopped : BOOL ;	//Motor is stopped
   StStarting : BOOL ;	//Motor is starting
   StStarted : BOOL ;	//Motor is started forward: Next Element can start
   StStopping : BOOL ;	//Motor is stopping
   StFault : BOOL ;	//Machine has a fault
   StClearing : BOOL ;	//Clearing time running, Blower started
   StCleared : BOOL ;	//Clearing time end, Blower is started
   Par : STRUCT
    ParObjectNo : INT ;	//Is used for communication with PC
    ParWithBlowOff : BOOL ;	//With BlowOffValve
    ParSingleLine : BOOL ;	//Airlock A and B in same blowline
    ParBlowerExternal : BOOL ;	//Blower is external
    ParWithShutOffValves : BOOL ;	//With ShutOffValves
    ParWithDiverter : BOOL ;	//With Diverter Valve
    ParClearingTime : INT ;	//Clearing time target [0.1s]
    OutClearingTime : INT ;	//Actual clearing time [0.1s]
    spare : DINT ;	//
   END_STRUCT ;
  END_STRUCT ;	
END_TYPE

TYPE "GCS7_M_FB68_Data"	// UDT 20680
VERSION : 0.0
  STRUCT 	// Interface to maschine FB50
   StCode : INT ;	//State as code
   InEnableConveying : BOOL ;	//Automatic mode: Conveying requested
   InEnableFilling1 : BOOL ;	//Automatic mode: Filling vessel requested
   InEnableFilling2 : BOOL ;	//Automatic mode: Filling vessel requested
   InAirOk : BOOL ;	//Pressure air is ok, example blower is started
   InMinPressure : BOOL ;	//Pressure > empty pressure
   InMaxPressure : BOOL ;	//Pressure > maximum pressure: Stop fluidization valve
   InOverPressure : BOOL ;	//Pressure > over pressure: immediately blow off
   InBlowoffIsOpen : BOOL ;	//Blow-off valve is open
   CmdOff : BOOL ;	//Manual mode:Pulse to stop all elements immediately
   CmdConveying : BOOL ;	//Manual mode:Pulse to start conveying
   CmdNext : BOOL ;	//Pulse to start the element in automatic mode (see global flags)
   CmdFaultReset : BOOL ;	//Command to reset fault
   InLocal : BOOL ;	//1= Local mode (no fault by start with service switch)
   InManual : BOOL ;	//1= Manual/ 0=Automatic
   CmdFilling1 : BOOL ;	//Manual mode: Pulse to fill vessel 1
   CmdFilling2 : BOOL ;	//Manual mode: Pulse to fill vessel 2
   CmdPulsing : BOOL ;	//Manual mode: Pulsing ConvValve
   InNoRestdischarge : BOOL ;	//Only a part batch, no clearing step
   spare0402 : BOOL ;
   OutLoaded : BOOL ;	//Output: Product is in vessel
   OutFault : BOOL ;	//Output: Summary fault
   OutBlowoff : BOOL ;	//Request to open blowoff valve
   OutEnableBlower : BOOL ;	//Output: Enable running blower
   spare0407 : BOOL ;
   StStopped : BOOL ;
   StFilling : BOOL ;
   StConveying : BOOL ;
   StPulsing : BOOL ;
   spare0504 : BOOL ;
   StClearing : BOOL ;
   StCleared : BOOL ;
   Par : STRUCT
    ParObjectNo : INT ;	//Is used for communication with PC
    ParType2Vessel : BOOL ;
    ParWithRecycValve : BOOL ;	//With element
    ParWithOutletValve : BOOL ;	//With element
    ParDelayFluidTime : INT ;	//[0.1s] Delay time to open fluidization valve running
    ParMinConveyingTime : INT  := 100;	//[0.1s] Minimum conveying time
    ParPulseBothTime : INT  := 100;	//[0.1s] StPulsing: ConvValve and FluidValve are open
    ParPulseFluidOnlyTime : INT  := 100;	//[0.1s] StPulsing: Only FluidValve is open
    ParClearingTime : INT  := 100;	//[0.1s] Clearing time in step StClearing
    ParPulseCnt : INT  := 4;	//Number of pulses in StPulsing
    spare18 : INT ;
    spare20 : INT ;
    spare22 : INT ;
    OutDelayFluidTime : INT ;
    OutConveyingTime : INT ;
    OutPulseTime : INT ;
    OutPulseCnt : INT ;
    OutClearingTime : INT ;
    OutDelayFluidDone : BOOL ;	//ParDelayFluidTime is done
    OutConvTimeDone : BOOL ;	//ParMinConveyingTime is done
    OutPulseFluidOnly : BOOL ;	//ParPulseFluidOnlyTime is running
    OutManFilling1 : BOOL ;	//Manual mode filling vessel 1
    OutManFilling2 : BOOL ;	//Manual mode filling vessel 2
    spare : INT ;
   END_STRUCT ;
  END_STRUCT ;	
END_TYPE

TYPE "GCS7_M_FB69_Data"	// UDT 20690
VERSION : 0.0
  STRUCT 	// Interface to maschine FB50
   StCode : INT ;	//State as code
   InEnable : BOOL ;	//Enable to run the motor
   spare0201 : BOOL ;	//Previous LS has been touched. Set by time interruted OB
   InUsed : BOOL ;	//Free for user: machine is used for active receiver
   spare0203 : BOOL ;
   spare0204 : BOOL ;
   spare0205 : BOOL ;
   spare0206 : BOOL ;
   spare0207 : BOOL ;
   CmdOff : BOOL ;	//Pulse to stop the machine in manual mode
   CmdOn : BOOL ;	//Pulse to start the machine in manual mode
   CmdNext : BOOL ;	//Pulse to start the element in automatic mode
   CmdFaultReset : BOOL ;	//Command to reset fault
   InLocal : BOOL ;	//1= Local mode (no fault by start with service switch)
   InManual : BOOL ;	//1= Manual/ 0=Automatic
   CmdPrevPos : BOOL ;	//Manual mode:Pulse move to previous position
   CmdNextPos : BOOL ;	//Manual mode:Pulse move to next position
   OutRev : BOOL ;	//Internal used: Find lower position
   OutFlagAdjusted : BOOL ;	//Internal used: Flag adusted
   OutFlagChange : BOOL ;	//Internal used: Change direction
   spare0403 : BOOL ;
   spare0404 : BOOL ;
   spare0405 : BOOL ;
   spare0406 : BOOL ;
   spare0407 : BOOL ;
   StStopped : BOOL ;	//Motor is stopped, in any position, not target position
   StAdjusting : BOOL ;	//Motor is running forward or reverse
   StAdjusted : BOOL ;	//Motor is stopped, not in target position
   StNoPosition : BOOL ;	//Motor is stopped, not in any position
   StFault : BOOL ;	//Machine has a fault
   InSetPos : ARRAY  [1 .. 32 ] OF //Target position
   BOOL ;
   InpLSPos : ARRAY  [1 .. 32 ] OF //LS position
   BOOL ;
   OutSetPos : ARRAY  [1 .. 32 ] OF //Target position
   BOOL ;
   InBinTarget : INT ;	//Only for SCADA system: Free for user
   InBinActual : INT ;	//Only for SCADA system: Free for user
   spare22 : INT ;	//Free for user
   Par : STRUCT
    ParObjectNo : INT ;	//Is used for communication with PC
    Par2Dir : BOOL ;	//Two direction
    ParNoOfPosition : INT  := 32;	//Number of positions
    spare : INT ;
   END_STRUCT ;
  END_STRUCT ;	
END_TYPE

TYPE "GCS7_M_FB81_Data"	// UDT 20810
VERSION : 0.0
  STRUCT 	// Interface to maschine FB50
   StCode : INT ;	//State as code
   InEnable : BOOL ;	//Enable to run the machine
   InClearing : BOOL ;	//Stop all motors after clearing time
   InpAirMinus : BOOL ;	//Close Air flap
   InpAirPlus : BOOL ;	//Open air flap
   InpFeedMinus : BOOL ;	//Close flap feedroll
   InpFeedPlus : BOOL ;	//Open flap feedroll
   CmdNewJob : BOOL ;	//New job
   InModeWarning : BOOL ;	//Flowdetector as Warning
   CmdOff : BOOL ;	//Pulse to stop the machine in manual mode
   CmdOn : BOOL ;	//Pulse to start machine in manual mode
   CmdNext : BOOL ;	//Pulse to start the element in automatic mode
   CmdFaultReset : BOOL ;	//Command to reset fault
   InLocal : BOOL ;	//1= Local mode (no fault by start with service switch)
   InManual : BOOL ;	//1= Manual/ 0=Automatic
   InAirRegulation : BOOL ;	//1=Automatic regualtion or AirFlap
   InSeqStop : BOOL ;	//Stop automatically after idling time
   OutStartReqMan : BOOL ;	//Start request in manaul mode
   OutFlapAirLocal : BOOL ;	//Position has been modified local
   OutFlapFeedLocal : BOOL ;	//Position has been modified local
   OutWarning : BOOL ;	//Warning from flow detector
   OutCleared : BOOL ;	//Clearing time Done
   spare0405 : BOOL ;
   spare0406 : BOOL ;
   spare0407 : BOOL ;
   StStopped : BOOL ;	//Machine is stopped
   StStarting : BOOL ;	//Machine is starting
   StStarted : BOOL ;	//Machine is started
   StStopping : BOOL ;	//Machine is stopping
   StFault : BOOL ;	//Machine has a fault
   StClearing : BOOL ;	//Clearing time is running
   InPosFlapAirNom : INT ;	//Target maximum position [0.0 .. 90.0°]
   InPosFlapAirMin : INT ;	//Target minimum position [0.0 .. 90.0°]
   InPosFlapFeed : INT ;	//Target position [0.0 .. 90.0°]
   InPosFlapLower : INT ;	//Target position [1,2,3]
   InPosFlapUpper : INT ;	//Target position [1,2,3]
   InLimitOverflowFault : INT ;	//Limit product overflow for fault [0.1%]
   InTolOverflow : INT ;	//Tolerance product overflow[0.1%]
   InOverflow : INT ;	//Nominal product overflow [0.1%]
   spare22 : INT ;
   OutPosFlapAir : INT ;	//Actual position [0.0 .. 90.0°]
   OutPosFlapFeed : INT ;	//Actual position [0.0 .. 90.0°]
   OutOverflow : INT ;	//Actual product overflow [0.1%]
   Par : STRUCT
    ParObjectNo : INT ;	//Is used for communication with PC
    ParWithVentus : BOOL  := TRUE;	//With Ventus
    ParWithSieve : BOOL  := TRUE;	//With Sieve
    ParWithFan2 : BOOL  := TRUE;	//With element Fan2
    ParWithFlapAir : BOOL  := TRUE;	//With element FlapAir
    ParWithFlapFeed : BOOL  := TRUE;	//With element FlapFeed
    ParWithFlowdetector : BOOL  := TRUE;	//With element Flowdetector
    ParWithFlapLower : BOOL ;	//With element FlapLower
    ParWithFlapUpper : BOOL ;	//With element FlapUpper
    ParClearingTime : INT ;	//Clearing time by deselect motor befor stop [0.1s]
    ParTI : INT  := 100;	//Time for integral regulator air flap [0.1s]
    spare : INT ;
    spare1 : INT ;
    spare2 : INT ;
    spare3 : INT ;
    spare4 : INT ;
    OutClearingTime : INT ;	//Actual clearing time [0.1s]
    OutPosFlapAirNom : REAL ;	//Actual target position [0.0 .. 90.0°]
    tmpPosFlapAir : INT ;	//Target position [0..100%]
    tmpPosFlapFeed : INT ;	//Target position [0..100%]
    tmpEdgeInpLocal : BOOL ;	//Positve edge push button
    spare281 : BOOL ;	//
   END_STRUCT ;
  END_STRUCT ;	
END_TYPE

TYPE "GCS7_M_FB82_Data"	// UDT 20820
VERSION : 0.0
  STRUCT 	// Interface to maschine FB50
   StCode : INT ;	//State as code
   InEnable : BOOL ;	//Automatic mode: Enable to run blower
   InEnableFilling : BOOL ;	//Automatic mode: Filling vessel requested
   InClearing : BOOL ;	//Automatic mode: Stop Conveying
   InNoWaitMinP : BOOL ;	//Not waiting for minimum pressure during clearing
   spare0204 : BOOL ;
   spare0205 : BOOL ;
   spare0206 : BOOL ;
   spare0207 : BOOL ;
   CmdOff : BOOL ;	//Manual mode:Pulse to stop all elements immediately
   CmdConveying : BOOL ;	//Manual mode:Pulse to start conveying
   CmdNext : BOOL ;	//Pulse to start the element in automatic mode (see global flags)
   CmdFaultReset : BOOL ;	//Command to reset fault
   InLocal : BOOL ;	//1= Local mode (no fault by start with service switch)
   InManual : BOOL ;	//1= Manual/ 0=Automatic
   CmdFilling : BOOL ;	//Manual mode: Pulse to fill vessel
   InSeqStop : BOOL ;	//Sequence stop
   OutWarning : BOOL ;	//Output: Pressure.OutNoMinP
   OutLoaded : BOOL ;	//Output: Product is in vessel
   OutAutostart : BOOL ;	//Autostart automatic mode
   spare0403 : BOOL ;
   OutPulseOn : BOOL ;	//(*1) During Clearing Time : Pulse Time On is running
   OutConveyingTimeDone : BOOL ;	//ParMinConveyingTime is done
   OutManFilling : BOOL ;	//Manual mode filling vessel
   OutManConveying : BOOL ;	//Manual mode conveying
   StStopped : BOOL ;
   StStarting : BOOL ;
   StConveying : BOOL ;
   StStopping : BOOL ;
   StFault : BOOL ;
   StClearing : BOOL ;
   StWaiting : BOOL ;
   StFilling : BOOL ;
   Par : STRUCT
    ParObjectNo : INT ;	//Is used for communication with PC
    ParWithFillingFlap : BOOL ;	//With element
    spare2_1 : BOOL ;
    spare2_2 : BOOL ;
    spare2_3 : BOOL ;
    spare4 : INT ;
    ParMinConveyingTime : INT  := 100;	//[0.1s] Minimum conveying time
    ParClearingTime : INT  := 100;	//[0.1s] Clearing time in step StClearing
    ParClearingPulseOn : INT  := 20;	//(*1) During Clearing Time: Fluidlift Valve pusling: Pulse Time On
    ParClearingPulseOff : INT  := 20;	//(*1) During Clearing Time : Fluidlift Valve pusling: Pulse Time Off
    spare14 : INT ;
    OutPulseTime : INT ;	//Actual pulsing time during clearing
    OutConveyingTime : INT ;
    OutClearingTime : INT ;
    spare : INT ;
   END_STRUCT ;
  END_STRUCT ;	
END_TYPE

TYPE "GCS7_FB84_Communication"	// UDT 20849
VERSION : 0.1
  STRUCT
   InMonCovered : BOOL ;	//After t4 must be in StCovered, otherwise it is a process fault
   InMonUncovered : BOOL ;	//After t5 must be in StUncovered, otherwise it is a process fault
   InPreAlarmCovered : BOOL ;	//LOG Pre-alarm if level is not covered
   InPreAlarmUncovered : BOOL ;	//LOG Pre-alarm if level is not uncovered
   InStopCoveredTime : BOOL ;	//Stop delay time t2
   InStopUncoveredTime : BOOL ;	//Stop delay time t3
   InpCovered : BOOL ;	//Digital input: 1=Covered , 0=Uncovered
   InpFaultDev : BOOL ;	//Digital input: fault device
   CmdRstCoveredTime : BOOL ;	//Restart delay time changing from Uncovered to Covered (t2)
   CmdRstUncoveredTime : BOOL ;	//Restart delay time changing from Covered to Uncovered (t3)
   CmdRunTimeoutTime : BOOL ;	//Run timeout time (only 1 working condition)
   CmdFaultReset : BOOL ;	//Command to reset fault
   InLocal : BOOL ;	//1= Local mode (automatic fault reset)
   spare0305 : BOOL ;
   InReport : BOOL ;	//Report of all state transitions
   OutTimeoutTime : BOOL ;	//Timeout time 1 working condition active
   InHWStop : BOOL ;	//HW stop is detected, no fault
   InDPFault : BOOL ;	//DP-Fault is detected, no fault
   OutPreAlarmCovered : BOOL ;	//Flag PreAlarmCovered is done
   OutPreAlarmUncovered : BOOL ;	//Flag PreAlarmUnCovered is done
   OutFlagPos : BOOL ;	//Positive flag InpCovered
   OutFlagNeg : BOOL ;	//Negative flag InpCovered
   OutpFaultReset : BOOL ;	//Reset alarm
   OutCovered : BOOL ;	//Copy of input signal
   StUncovered : BOOL ;	//Level is uncovered, delay time finished, monitoring is off
   StCtoCovered : BOOL ;	//Changing to Covered
   StCovered : BOOL ;	//Level is Covered, delay time finished
   StCtoUncovered : BOOL ;	//Changing to Uncovered
   StFault : BOOL ;	//Signal has not requested value, monitoring is active
  END_STRUCT ;	
END_TYPE

TYPE "GCS7_FB85_Data"	// UDT 20850
VERSION : 0.0
  STRUCT 	// Interface to maschine FB50
   StCode : INT ;	//State as code
   InEnableDown : BOOL ;	//Enable to move downwards
   InEnableUp : BOOL ;	//Enable to move upwards
   InInterlocked : BOOL ;	//Interlocked mode
   InPowerOk : BOOL ;	//Power is ok
   InPowerOkDelayDone : BOOL ;	//Delay time power ok is done
   InUnloading : BOOL ;	//Moving with pulsing
   InCalibration : BOOL ;	//Calibration mode
   InCalibrationZero : BOOL ;	//Setting to zero point in calibration mode
   CmdOff : BOOL ;	//Pulse to stop motor immediately in manual mode
   CmdUp : BOOL ;	//Pulse to start upwards in manual mode
   CmdNext : BOOL ;	//Pulse to start the element in automatic mode
   CmdFaultReset : BOOL ;	//Command to reset fault
   InLocal : BOOL ;	//1= Local mode (no fault by start with service switch)
   InManual : BOOL ;	//1= Manual/ 0=Automatic
   CmdDown : BOOL ;	//Pulse to start downwards in manual mode
   InEnableLowerMinPos : BOOL ;	//Enable to move downwards < minimum position
   OutAdjustedLeft : BOOL ;	//Left side is adjusted
   OutAdjustedRight : BOOL ;	//Right side is adjusted
   OutPositionLeftToHigh : BOOL ;	//Left motor must stop until both side are on same level
   OutPositionRightToHigh : BOOL ;	//Left motor must stop until both side are on same level
   OutDifferenceFault : BOOL ;	//Difference to high, stop both motor
   OutHigherMinPos : BOOL ;	//Actual position > minimum position
   OutPulseOn : BOOL ;	//Pulsing: Pulse On
   spare47 : BOOL ;	//
   StStopped : BOOL ;	//Motors are stopped
   StStarting : BOOL ;	//Motors are starting
   StStartedUP : BOOL ;	//Motors is started in upwards
   StStopping : BOOL ;	//Motors are stopping
   StFault : BOOL ;	//Machine has a fault
   StStartedDown : BOOL ;	//Machine is started downwards
   StAdjusted : BOOL ;	//Machine is enabled and in target psoition
   spare57 : BOOL ;	//
   OutManStartReqDown : BOOL ;	//Manual Mode Start request downwards
   OutManStartReqUp : BOOL ;	//Manual Mode Start request upwards
   InPositionTarget : INT ;	//Target position in [mm]
   OutPositionLeft : INT ;	//Actual position left in [mm]
   OutPositionRight : INT ;	//Actual position right in [mm]
   OutPositionDifference : INT ;
   OutIncrementLeft : DINT ;	//Copy of 32Bit from incremental counter left side
   OutIncrementRight : DINT ;	//Copy of 32Bit from incremental counter right side
   OutPulseTime : INT ;	//Actual Pulse Time [0.1s]
   BankingLoadingScrew : INT ;	//Banking screw bei laoding
   spare3 : INT ;
   spare4 : INT ;
   spare5 : INT ;
   spare6 : INT ;
   spare7 : INT ;
   spare8 : INT ;
   spare9 : INT ;
   Par : STRUCT
    ParObjectNo : INT ;	//Is used for communication with PC
    spare : BOOL ;
    ParPositionTopLeftInc : INT  := 693;	//Position Top Left [Increments]
    ParPositionTopRightInc : INT  := 690;	//Position Top Right [Increments]
    ParPositionTopLeftUnits : INT  := 1665;	//Position Top Left [mm]
    ParPositionTopRightUnits : INT  := 1665;	//Position Top Right [mm]
    ParPositionMin : INT ;	//Minimum Psoition [mm]
    ParTolPosition : INT ;	//Tolerance for target position [mm]
    ParMaxOffTrackPause : INT ;	//Maximum off-track before one motor must stop [mm]
    ParMaxOffTrackFault : INT ;	//Maximum off-track before machine changes to fault [mm]
    ParMonTime : INT  := 50;	//t0 Monitoring time for moving [0.1s]
    ParIOByteNoCounterLeft : INT ;	//First byte of IO of counter module left side
    ParIOByteNoCounterRight : INT ;	//First byte of IO of counter module right side
    OutMonTimeLeft : INT ;	//Monitoring time left side
    OutMonTimeRight : INT ;	//Monitoring time right side
    OutUnitsPerIncLeft : REAL ;	//Number of [mm] per increment
    OutUnitsPerIncRight : REAL ;	//Number of [mm] per increment
    ParPulseOnTime : INT ;	//Pulse lenght time [0.1s]
    ParPulseOffTime : INT ;	//Pausing time between to pulses [0.1s]
    spare3 : INT ;
    spare4 : INT ;
    spare5 : INT ;
   END_STRUCT ;
  END_STRUCT ;	
END_TYPE

TYPE "GCS7_FB85_Counter"	// UDT 20851
VERSION : 0.0
  STRUCT 	// Interface to maschine FB50
   OutpSetCount : DWORD ;	//de:Ladewert des 1Count24V/100kHz
   OutpSW_GATE : BOOL ;	//de:Steuerbit SW-Tor
   OutpCTRL_SYN : BOOL ;	//de:Freigabe Synchronisation
   OutpRES_STS : BOOL ;	//de:Anstoß Rücksetzen Statusbit
   OutpSET_DO1 : BOOL ;	//de:Steuerbit DO1
   OutpCTR_DO1 : BOOL ;	//de:Freigabe DO1
   OutpSET_DO2 : BOOL ;	//de:Steuerbit DO2
   OutpCTR_DO2 : BOOL ;	//de:Freigabe DO2
   OutpEXTF_ACK : BOOL ;	//de:Diagnosefehlerquittung
   OutpLOAD_VAL : BOOL ;	//de:Zähler direkt laden
   OutpLOAD_PREPARE : BOOL ;	//de:Zähler vorbereitend laden
   OutpCMP_VAL1 : BOOL ;	//de:Vergleichswert 1 laden
   OutpCMP_VAL2 : BOOL ;	//de:Vergleichswert 2 laden
   OutpC_DOPARAM : BOOL ;	//de:Funktion und Verhalten von DO1, DO2 ändern
   OutpSpare65 : BOOL ;	//de:Reserve = 0
   OutpSpare66 : BOOL ;	//de:Reserve = 0
   OutpSpare67 : BOOL ;	//de:Reserve = 0
   OutpTrack_A : BOOL ;	//de:Reserve = 0
   OutpTrack_A_pos_Flag : BOOL ;	//de:Reserve = 0
   OutpTrack_B : BOOL ;	//de:Reserve = 0
   OutpTrack_B_pos_Flag : BOOL ;	//de:Reserve = 0
   OutpSpare74 : BOOL ;	//de:Reserve = 0
   OutpSpare75 : BOOL ;	//de:Reserve = 0
   OutpSpare76 : BOOL ;	//de:Reserve = 0
   OutpSpare77 : BOOL ;	//de:Reserve = 0
   OutpSpare8 : BYTE ;	//de:Reserve = 0
   InpActCount : DWORD ;	//de:Aktueller Zählwert
   InpSTS_LOAD : BOOL ;	//de:Ladefunktion läuft
   InpERR_LOAD : BOOL ;	//de:Fehler bei Ladefunktion
   InpRES_STS_A : BOOL ;	//de:Rücksetzen der Statusbit läuft
   InpSpare53 : BOOL ;	//de:Reserve = 0
   InpSpare54 : BOOL ;	//de:Reserve = 0
   InpERR_PARA : BOOL ;	//de:Parametrierfehler
   InpERR_DO1 : BOOL ;	//de:Kurzschluss / Drahtbruch / Übertemperatur
   InpERR_24V : BOOL ;	//de:Kurschluss Geberversorgung
   InpSTS_GATE : BOOL ;	//de:Status internes Tor
   InpSTS_DI : BOOL ;	//de:Status DI
   InpSpare62 : BOOL ;	//de:Reserve = 0
   InpSTS_DO1 : BOOL ;	//de:Status DO1
   InpSTS_DO2 : BOOL ;	//de:Status DO2
   InpSpare65 : BOOL ;	//de:Reserve = 0
   InpSTS_C_UP : BOOL ;	//de:Status Richtung vorwärts
   InpSTS_C_DN : BOOL ;	//de:Status Richtung rückwärts
   InpSTS_SYN : BOOL ;	//de:Status Synchronisation
   InpSpare71 : BOOL ;	//de:Reserve = 0
   InpSpare72 : BOOL ;	//de:Reserve = 0
   InpSTS_CMP1 : BOOL ;	//de:Status Vergleicher 1
   InpSTS_CMP2 : BOOL ;	//de:Status Vergleicher 2
   InpSTS_OFWL : BOOL ;	//de:Obere Zählgrenze
   InpSTS_UFWL : BOOL ;	//de:Untere Zählgrenze
   InpSTS_ND : BOOL ;	//de:Nulldurchgang im Zählbereich bei Zählen ohne Hauptzählrichtung
   InpSpare8 : BYTE ;	//de:Reserve = 0
   VarInpHold : DWORD ;	//Internal used to restor counter value after power fault
  END_STRUCT ;	
END_TYPE

TYPE "GCS7_FB86_Data"	// UDT 20860
VERSION : 0.0
  STRUCT 	// Interface to maschine FB50
   StCode : INT ;	//State as code
   InEnableRev : BOOL ;	//Enable to run machine reverse
   InEnableFwd : BOOL ;	//Enable to run machine forward
   InInterlocked : BOOL ;	//Interlocked mode
   InPowerOk : BOOL ;	//Power is ok
   InPowerOkDelayDone : BOOL ;	//Delay time power ok is done
   CmdNewJob : BOOL ;	//Set OutCntRound=0, Set OutStartPosition
   InAdjusting : BOOL ;	//1=Adjusting 0=Endless
   InLoading : BOOL ;	//1=Loging is active
   CmdOff : BOOL ;	//Pulse to stop motor immediately in manual mode
   CmdOnFwd : BOOL ;	//Pulse to start forward in manual mode
   CmdNext : BOOL ;	//Pulse to start the element in automatic mode
   CmdFaultReset : BOOL ;	//Command to reset fault
   InLocal : BOOL ;	//1= Local mode (no fault by start with service switch)
   InManual : BOOL ;	//1= Manual/ 0=Automatic
   CmdOnRev : BOOL ;	//Pulse to start reverse in manual mode
   spare37 : BOOL ;	//
   CmdSetZeroPoint : BOOL ;	//Set Counter modul to 0
   OutAdjusted : BOOL ;	//Machine is adjusted in target position
   OutEdgeLoading : BOOL ;	//Internal used to generate alarm when Flowdetector is covered at start
   OutEdgeCntRoundFwd : BOOL ;	//Internal used to count round
   OutEdgeCntRoundRev : BOOL ;	//Internal used to count round
   spare45 : BOOL ;	//
   spare46 : BOOL ;	//
   spare47 : BOOL ;	//
   StStopped : BOOL ;	//Motors are stopped
   StStarting : BOOL ;	//Motors are starting
   StStartedFwd : BOOL ;	//Motors is started in upwards
   StStopping : BOOL ;	//Motors are stopping
   StFault : BOOL ;	//Machine has a fault
   StStartedRev : BOOL ;	//Machine is started downwards
   StAdjusted : BOOL ;	//Machine is enabled and in target psoition
   spare57 : BOOL ;	//
   OutManStartReqRev : BOOL ;	//Manual Mode Start request reverse
   OutManStartReqFwd : BOOL ;	//Manual Mode Start request forward
   VarDetaGrt170 : BOOL ;	//Internal used for round counter: Delta angle > 170 °
   InPositionTarget : INT ;	//Target position in [0.1°]
   InSpeed : INT ;	//Target speed [0.01%]
   OutPositionAngle : INT ;	//Actual position in [0.1°]
   OutPositionRel : INT ;	//Actual position in [0.1%]
   OutCntRound : DINT ;	//Actual numbers of round
   OutIncrement : DINT ;	//Copy 32Bit from incremental counter
   OutPositionStart : INT ;	//Start position for round counter
   spare1 : DINT ;
   spare2 : DINT ;
   spare3 : DINT ;
   spare4 : DINT ;
   spare5 : DINT ;
   spare6 : DINT ;
   spare7 : DINT ;
   Par : STRUCT
    ParObjectNo : INT ;	//Is used for communication with PC
    ParEndless : BOOL ;	//Endless rotation
    ParIncrementsPerRound : DINT ;	//Number of increment per round (360°)
    ParTolPosition : INT ;	//Tolerance for target position [0.1°]
    ParMonTime : INT ;	//t0 Monitoring time for moving [0.1s]
    ParIOByteNoCounter : INT ;	//First byte of IO of counter module
    OutMonTime : INT ;	//Monitoring time left side
    spare1 : DINT ;
    spare2 : INT ;
    spare3 : INT ;
    spare4 : INT ;
   END_STRUCT ;
  END_STRUCT ;	
END_TYPE

TYPE "GCS7_M_FB87_Data"	// UDT 20870
VERSION : 0.0
  STRUCT 	// Interface to maschine FB50
   StCode : INT ;	//State as code
   InEnable : BOOL ;	//Enable to run machine
   InDisableSide1 : BOOL ;	//Side1 not used
   InDisableSide2 : BOOL ;	//Side2 not used
   InOverrideHL : BOOL ;	//Override HL
   InEnableDosing : BOOL ;	//Enable Dosing for MDDR/T
   InRestDischarge : BOOL ;	//Restdischarge
   InpPressureSide1 : BOOL ;	//1=Working pressure rolls
   InpPressureSide2 : BOOL ;	//1=Working pressure rolls
   CmdOff : BOOL ;	//Pulse to start the element immediately (manual mode)
   CmdOn : BOOL ;	//Pulse to stop  the element immediately (manual mode)
   CmdNext : BOOL ;	//Pulse to start the element in automatic mode
   CmdFaultReset : BOOL ;	//Command to reset fault
   InLocal : BOOL ;	//1= Local mode (no fault by start with service switch)
   InManual : BOOL ;	//1= Manual/ 0=Automatic
   spare3 : BOOL ;
   InSeqStop : BOOL ;	//Sequence stop
   OutStartupDone : BOOL ;
   OutStartMan : BOOL ;	//Internal used
   OutWarning : BOOL ;	//Warning
   spare5 : BOOL ;
   spare6 : BOOL ;
   spare7 : BOOL ;
   spare8 : BOOL ;
   spare9 : BOOL ;
   StStopped : BOOL ;
   StStarting : BOOL ;
   StStarted : BOOL ;
   StStopping : BOOL ;
   StFault : BOOL ;
   StEngaged : BOOL ;
   Par : STRUCT
    ParObjectNo : INT ;	//Is used for communication with PC
    spare1 : INT ;
    ParWithHLInletSide1 : BOOL  := TRUE;	//HL Inlet side 1 (if divided then right passage of side 1)
    ParWithHLInletSide2 : BOOL  := TRUE;	//HL Inlet side 2 (if divided then right passage of side 2)
    ParWithSMSide1 : BOOL ;	//With speedmonitor side 1
    ParWithSMSide2 : BOOL ;	//With speedmonitor side 2
    ParManual : BOOL ;	//No interlocking in maual mode
    Par4Rolls : BOOL ;	//4 roll stand
    ParWithMDDx : BOOL ;	//Probfibus interface to MDDR/T
    ParWithHLInletSide1Div : BOOL ;	//Level Inlet left passage of side 1
    ParWithHLInletSide2Div : BOOL ;	//Level Inlet left passage of side 2
    ParWithMotorUpSide1 : BOOL  := TRUE;	//Only used roll stand with 8 rolls
    ParWithMotorUpSide2 : BOOL  := TRUE;	//Only used roll stand with 8 rolls
    ParWithHLOutlet1Side1 : BOOL  := TRUE;	//1st HL Outlet side 1
    ParWithHLOutlet2Side1 : BOOL  := TRUE;	//2nd HL Outlet side 1
    ParWithHLOutlet1Side2 : BOOL  := TRUE;	//1st HL Outlet side 2
    ParWithHLOutlet2Side2 : BOOL  := TRUE;	//2nd HL Outlet side 2
    ParWithHLOutlet3Side1 : BOOL ;	//3th HL Outlet side 1
    ParWithHLOutlet3Side2 : BOOL ;	//3th HL Outlet side 2
   END_STRUCT ;
  END_STRUCT ;	
END_TYPE

TYPE "GCS7_M_FB88_Data"	// UDT 20880
VERSION : 0.0
  STRUCT 	// Interface to maschine FB50
   StCode : INT ;	//State as code
   InEnable : BOOL ;	//Enable to run the motor reverse
   InRestDischarge : BOOL ;	//Rest discharge of the bin
   spare0202 : BOOL ;	//Disable Vibro
   spare0203 : BOOL ;
   spare0204 : BOOL ;
   InDoorClosed : BOOL ;	//Door is closed
   InDoorOpen : BOOL ;	//Door is opend
   spare0207 : BOOL ;
   CmdOff : BOOL ;	//Pulse to start the element immediately (manual mode)
   CmdOn : BOOL ;	//Pulse to stop  the element immediately (manual mode)
   CmdNext : BOOL ;	//Pulse to start the element in automatic mode
   CmdFaultReset : BOOL ;	//Command to reset fault
   InLocal : BOOL ;	//1= Local mode (no fault by start with service switch)
   InManual : BOOL ;	//1= Manual/ 0=Automatic
   spare0306 : BOOL ;
   spare0307 : BOOL ;
   OutEnableConveying : BOOL ;	//Enable for Conveying
   spare0401 : BOOL ;
   spare0402 : BOOL ;
   spare0403 : BOOL ;
   spare0404 : BOOL ;
   spare0405 : BOOL ;
   spare0406 : BOOL ;
   spare0407 : BOOL ;
   StStopped : BOOL ;	//Discharger is closed
   StStarting : BOOL ;	//Discharger is opening
   StStarted : BOOL ;	//Discharger is open
   StStopping : BOOL ;	//Discharger is closing
   StFault : BOOL ;	//Machine has a fault
   Par : STRUCT
    ParObjectNo : INT ;	//Is used for communication with PC
    ParWithSlide1 : BOOL ;	//With element
    ParWithSlide2 : BOOL ;	//With element
    ParWithSlide3 : BOOL ;	//With element
    ParWithSlide4 : BOOL ;	//With element
    spare10 : INT ;
    spare12 : INT ;
    spare14 : INT ;
    spare16 : INT ;
    spare18 : INT ;
   END_STRUCT ;
  END_STRUCT ;	
END_TYPE

TYPE "SSW_EL_ASI_Slave"	// UDT 28995
VERSION : 0.1
  STRUCT
   Par : STRUCT
    ParDIDO : BOOL ;
    ParAI : BOOL ;
    ParAO : BOOL ;
   END_STRUCT ;
   StCode : INT ;
   OutDetected : BOOL ;	//1= Detected Slaves A (Read with 0x46)
   OutCfgDiff : BOOL ;	//1= Slaves A with configuartion diff.(Read with 0x57)
   OutPeripheralFault : BOOL ;	//1= Slaves A peripheral failure (Read with 0x3E)
   OutCorrupted : BOOL ;	//1= Corrupped Slaves A (Read with 0x6C)
   Spare44 : BOOL ;
   Spare45 : BOOL ;
   Spare46 : BOOL ;
   OutMsgDone : BOOL ;	//LOG Message Done
   StOk : BOOL ;	//1= Slave ok
   StFault : BOOL ;	//1= Slave is Faulted
   OutResult : INT ;	//Result Value of Mailbox communication
   Ch1 : INT ;
   Ch2 : INT ;
   Ch3 : INT ;
   Ch4 : INT ;
  END_STRUCT ;	
END_TYPE

TYPE "ASW_UDTOnOffCmd"	// UDT 32700
VERSION : 0.0
  STRUCT 	//Function key for CWA
   Cmd08 : BOOL ;	//Not used
   Cmd09 : BOOL ;	//Not used
   Cmd10 : BOOL ;	//Not used
   Cmd11 : BOOL ;	//Not used
   Cmd12 : BOOL ;	//Not used
   Cmd13 : BOOL ;	//Not used
   Cmd14 : BOOL ;	//Not used
   Cmd15 : BOOL ;	//Not used
   CmdPulse00OverrideLL : BOOL ;	//Override sender low levels
   CmdPulse01 : BOOL ;	//Not used
   CmdPulse02 : BOOL ;	//Not used
   CmdPulse03 : BOOL ;	//Not used
   CmdPulse04 : BOOL ;	//Not used
   CmdPulse05 : BOOL ;	//Not used
   CmdPulse06 : BOOL ;	//Not used
   CmdPulse07 : BOOL ;	//Not used
  END_STRUCT ;	
END_TYPE

TYPE "ASW_UDTSecNom"	// UDT 32701
VERSION : 0.0
  STRUCT 	//Function key for CWA
   Par1On : STRUCT 	//Job parameters
    Cmd08 : BOOL ;	//Not used
    Cmd09 : BOOL ;	//Not used
    Cmd10 : BOOL ;	//Not used
    Cmd11 : BOOL ;	//Not used
    Cmd12 : BOOL ;	//Not used
    Cmd13 : BOOL ;	//Not used
    Cmd14 : BOOL ;	//Not used
    Cmd15 : BOOL ;	//Not used
    Cmd00 : BOOL ;	//Not used
    Cmd01 : BOOL ;	//Not used
    Cmd02 : BOOL ;	//Not used
    Cmd03 : BOOL ;	//Not used
    Cmd04 : BOOL ;	//Not used
    Cmd05 : BOOL ;	//Not used
    Cmd06 : BOOL ;	//Not used
    Cmd07 : BOOL ;	//Not used
   END_STRUCT ;
   Par2On : STRUCT 	//Job parameters
    Cmd08 : BOOL ;	//Not used
    Cmd09 : BOOL ;	//Not used
    Cmd10 : BOOL ;	//Not used
    Cmd11 : BOOL ;	//Not used
    Cmd12 : BOOL ;	//Not used
    Cmd13 : BOOL ;	//Not used
    Cmd14 : BOOL ;	//Not used
    Cmd15 : BOOL ;	//Not used
    Cmd00 : BOOL ;	//Not used
    Cmd01 : BOOL ;	//Not used
    Cmd02 : BOOL ;	//Not used
    Cmd03 : BOOL ;	//Not used
    Cmd04 : BOOL ;	//Not used
    Cmd05 : BOOL ;	//Not used
    Cmd06 : BOOL ;	//Not used
    Cmd07 : BOOL ;	//Not used
   END_STRUCT ;
   Par3On : STRUCT 	//Job parameters
    Cmd08 : BOOL ;	//Not used
    Cmd09 : BOOL ;	//Not used
    Cmd10 : BOOL ;	//Not used
    Cmd11 : BOOL ;	//Not used
    Cmd12 : BOOL ;	//Not used
    Cmd13 : BOOL ;	//Not used
    Cmd14 : BOOL ;	//Not used
    Cmd15 : BOOL ;	//Not used
    Cmd00 : BOOL ;	//Not used
    Cmd01 : BOOL ;	//Not used
    Cmd02 : BOOL ;	//Not used
    Cmd03 : BOOL ;	//Not used
    Cmd04 : BOOL ;	//Not used
    Cmd05 : BOOL ;	//Not used
    Cmd06 : BOOL ;	//Not used
    Cmd07 : BOOL ;	//Not used
   END_STRUCT ;
   Par4On : STRUCT 	//Job parameters
    Cmd08 : BOOL ;	//Not used
    Cmd09 : BOOL ;	//Not used
    Cmd10 : BOOL ;	//Not used
    Cmd11 : BOOL ;	//Not used
    Cmd12 : BOOL ;	//Not used
    Cmd13 : BOOL ;	//Not used
    Cmd14 : BOOL ;	//Not used
    Cmd15 : BOOL ;	//Not used
    Cmd00 : BOOL ;	//Not used
    Cmd01 : BOOL ;	//Not used
    Cmd02 : BOOL ;	//Not used
    Cmd03 : BOOL ;	//Not used
    Cmd04 : BOOL ;	//Not used
    Cmd05 : BOOL ;	//Not used
    Cmd06 : BOOL ;	//Not used
    Cmd07 : BOOL ;	//Not used
   END_STRUCT ;
   LineFlowrate : INT ;	//Line flowrate, for turnover only
   NotUsed1 : INT ;	//Not used
   NotUsed2 : WORD ;
   NotUsed3 : WORD ;
   NotUsed4 : WORD ;
   NotUsed5 : WORD ;
  END_STRUCT ;	
END_TYPE

TYPE "ASW_UDTSecAc"	// UDT 32702
VERSION : 0.0
  STRUCT 	//Function key for CWA
   Par1On : STRUCT 	//Job parameter status
    StaOn08 : BOOL ;	//Not used
    StaOn09 : BOOL ;	//Not used
    StaOn10 : BOOL ;	//Not used
    StaOn11 : BOOL ;	//Not used
    StaOn12 : BOOL ;	//Not used
    StaOn13 : BOOL ;	//Not used
    StaOn14 : BOOL ;	//Not used
    StaOn15 : BOOL ;	//Not used
    StaOn00 : BOOL ;	//Not used
    StaOn01 : BOOL ;	//Not used
    StaOn02 : BOOL ;	//Not used
    StaOn03 : BOOL ;	//Not used
    StaOn04 : BOOL ;	//Not used
    StaOn05 : BOOL ;	//Not used
    StaOn06 : BOOL ;	//Not used
    StaOn07 : BOOL ;	//Not used
   END_STRUCT ;
   Par2On : STRUCT 	//Job parameter status
    StaOn08 : BOOL ;	//Not used
    StaOn09 : BOOL ;	//Not used
    StaOn10 : BOOL ;	//Not used
    StaOn11 : BOOL ;	//Not used
    StaOn12 : BOOL ;	//Not used
    StaOn13 : BOOL ;	//Not used
    StaOn14 : BOOL ;	//Not used
    StaOn15 : BOOL ;	//Not used
    StaOn00 : BOOL ;	//Not used
    StaOn01 : BOOL ;	//Not used
    StaOn02 : BOOL ;	//Not used
    StaOn03 : BOOL ;	//Not used
    StaOn04 : BOOL ;	//Not used
    StaOn05 : BOOL ;	//Not used
    StaOn06 : BOOL ;	//Not used
    StaOn07 : BOOL ;	//Not used
   END_STRUCT ;
   Par3On : STRUCT 	//Job parameter status
    StaOn08 : BOOL ;	//Not used
    StaOn09 : BOOL ;	//Not used
    StaOn10 : BOOL ;	//Not used
    StaOn11 : BOOL ;	//Not used
    StaOn12 : BOOL ;	//Not used
    StaOn13 : BOOL ;	//Not used
    StaOn14 : BOOL ;	//Not used
    StaOn15 : BOOL ;	//Not used
    StaOn00 : BOOL ;	//Not used
    StaOn01 : BOOL ;	//Not used
    StaOn02 : BOOL ;	//Not used
    StaOn03 : BOOL ;	//Not used
    StaOn04 : BOOL ;	//Not used
    StaOn05 : BOOL ;	//Not used
    StaOn06 : BOOL ;	//Not used
    StaOn07 : BOOL ;	//Not used
   END_STRUCT ;
   Par4On : STRUCT 	//Job parameter status
    StaOn08 : BOOL ;	//Not used
    StaOn09 : BOOL ;	//Not used
    StaOn10 : BOOL ;	//Not used
    StaOn11 : BOOL ;	//Not used
    StaOn12 : BOOL ;	//Not used
    StaOn13 : BOOL ;	//Not used
    StaOn14 : BOOL ;	//Not used
    StaOn15 : BOOL ;	//Not used
    StaOn00 : BOOL ;	//Not used
    StaOn01 : BOOL ;	//Not used
    StaOn02 : BOOL ;	//Not used
    StaOn03 : BOOL ;	//Not used
    StaOn04 : BOOL ;	//Not used
    StaOn05 : BOOL ;	//Not used
    StaOn06 : BOOL ;	//Not used
    StaOn07 : BOOL ;	//Not used
   END_STRUCT ;
   ValueNotUsed5 : INT ;	//Not used
   ValueNotUsed6 : INT ;	//Not used
   ValueNotUsed7 : INT ;	//Not used
   ValueNotUsed8 : INT ;	//Not used
   ValueNotUsed9 : INT ;	//Not used
   ValueNotUsed10 : INT ;	//Not used
  END_STRUCT ;	
END_TYPE

